FUNCTION_BLOCK Simulator
VAR_INPUT
	CurrentValue : REAL;
	TargetValue : REAL;
END_VAR
VAR_OUTPUT
	SimulatedValue : REAL;
END_VAR
VAR
	random_value : LREAL;
	fb_ran : DRAND;
END_VAR

fb_ran(Seed := 0, Num => random_value);
random_value := 0.5 * STRING_TO_REAL(LREAL_TO_FMTSTR(random_value, 2, TRUE));
IF ABS(CurrentValue-TargetValue)>0.5 THEN
	IF CurrentValue < TargetValue THEN
		CurrentValue := CurrentValue + random_value;
	ELSE
		CurrentValue := CurrentValue - random_value;
	END_IF
END_IF
SimulatedValue := STRING_TO_REAL(LREAL_TO_FMTSTR(CurrentValue, 2, TRUE)); //Rounding again here to clear any errors above

END_FUNCTION_BLOCK

(* stored: Version 1.1.0.1, ProductVersion 3.1.4024.3
   POU Simulator: Id {6eb8117d-1313-4ef4-b546-5a777e3c37ab}, SpecialFunc None *)
